(* IEC 61131-3 sources: nvidia-ai-factory-controls/libraries/AIFactory_Communication/POUs/Subscribers, 5 files *)

(* ---- FB_Subscriber_BACnet.fb ---- *)
(* =============================================================================
    FB_Subscriber_BACnet — BACnet/IP Client Subscriber
    Common Library | NVIDIA AI Factory Controls
   =============================================================================

   PURPOSE:
     Implements I_DataSubscriber by reading BACnet objects from external
     BMS/HVAC controllers. Used to collect:
       • Ambient temperature from building sensors
       • Outdoor wet-bulb temperature (for economizer decisions)
       • HVAC status (AHU running, damper positions)
       • Chilled water supply temperature from central plant
       • Building fire alarm status (BACnet notification class)

   POLLING MODEL:
     Similar to Modbus subscriber: maintains a poll table of
     BACnet ReadProperty requests. Cycles through in round-robin.

   BACnet SERVICES USED:
     • ReadProperty (single object read)
     • ReadPropertyMultiple (batch read — more efficient)
     • SubscribeCOV (Change-of-Value subscription — event-driven)

   COV (Change-of-Value):
     For critical values (fire alarm, ambient temp), use COV subscription
     instead of polling. BACnet server pushes changes immediately.
     Reduces latency from poll-interval to near-real-time.

   REQUIRES:
     CODESYS BACnet/IP Client device in project tree.
     Or: BACnet client library.

   THREAD SAFETY:
     Runs in Communication_Task. BACnet I/O is handled by CODESYS
     BACnet stack asynchronously; this FB reads the results.
   ============================================================================= *)

(* ═══════════════════════════════════════════════════════════════════════════════
   DECLARATION
   ═══════════════════════════════════════════════════════════════════════════════ *)

FUNCTION_BLOCK FB_Subscriber_BACnet IMPLEMENTS I_DataSubscriber
VAR_INPUT
    (* --- Timing --- *)
    fCycleTime_s         : REAL := 0.1;
    nMaxPollsPerCycle    : USINT := 4;
    nStaleTimeout_ms     : UDINT := 10000;

    (* --- COV Configuration --- *)
    bUseCOV              : BOOL := TRUE;    (* Prefer COV over polling *)
    nCOV_Lifetime_s      : UDINT := 300;    (* COV subscription lifetime *)
END_VAR

VAR
    _bConnected          : BOOL;
    _nSubscriptionCount  : UDINT;
    _nStaleCount         : UDINT;

    (* --- Poll Request Table --- *)
    _astPollRequests     : ARRAY[1..32] OF ST_BACnetPollRequest;
    _nPollCount          : USINT;
    _nCurrentPoll        : USINT;

    (* --- COV Subscriptions --- *)
    _astCOV_Subs         : ARRAY[1..16] OF ST_BACnetCOVSub;
    _nCOV_Count          : USINT;

    (* --- Received Data --- *)
    _astReceivedData     : ARRAY[1..64] OF ST_Subscription;
    _nReceivedCount      : UINT;

    (* --- Discovered Values (commonly needed) --- *)
    fAmbientTemp         : REAL;            (* Outdoor ambient temperature [°C] *)
    fWetBulbTemp         : REAL;            (* Wet-bulb temperature [°C] *)
    fCHW_SupplyTemp      : REAL;            (* Chilled water supply [°C] *)
    bBuildingFireAlarm   : BOOL;            (* Building fire alarm active *)
    bAHU_Running         : ARRAY[1..4] OF BOOL;  (* Air handling unit status *)

    (* --- Statistics --- *)
    _nTotalReads         : UDINT;
    _nSuccessfulReads    : UDINT;
    _nCOV_Notifications  : UDINT;           (* COV events received *)

    (* --- Edge Triggers --- *)
    _rtrigFireAlarm      : R_TRIG;          (* Building fire alarm activated *)
    _ftrigFireAlarm      : F_TRIG;          (* Building fire alarm cleared *)
END_VAR

(* ═══════════════════════════════════════════════════════════════════════════════
   IMPLEMENTATION
   ═══════════════════════════════════════════════════════════════════════════════ *)

(* --- Fire Alarm Edge Detection --- *)
_rtrigFireAlarm(CLK := bBuildingFireAlarm);
_ftrigFireAlarm(CLK := bBuildingFireAlarm);

(* --- Round-Robin Polling (same pattern as Modbus subscriber) --- *)
(* In production with CODESYS BACnet library:
   FOR i := 1 TO nMaxPollsPerCycle DO
       _nCurrentPoll := _nCurrentPoll + 1;
       IF _nCurrentPoll > _nPollCount THEN _nCurrentPoll := 1; END_IF

       // Execute BACnet ReadProperty
       // Object: _astPollRequests[_nCurrentPoll].nObjectType
       // Instance: _astPollRequests[_nCurrentPoll].nObjectInstance
       // Property: Present_Value (85)

       // On success: store value, update timestamp
       // On error: increment error count
   END_FOR *)

(* --- COV Subscription Renewal --- *)
(* BACnet COV subscriptions expire. Renew before lifetime expires.
   In production: check each _astCOV_Subs lifetime remaining,
   re-subscribe if < 60 seconds remaining. *)

(* --- Stale Detection --- *)
_nStaleCount := 0;
(* Check all subscriptions for staleness *)

(* ---- FB_Subscriber_Modbus.fb ---- *)
(* =============================================================================
    FB_Subscriber_Modbus — Modbus TCP Master (Client) Subscriber
    Common Library | NVIDIA AI Factory Controls
   =============================================================================

   PURPOSE:
     Implements I_DataSubscriber by polling Modbus TCP slave devices.
     Used to collect data from:
       • Energy meters (Schneider PM5xxx, ABB M4M)
       • UPS systems (Vertiv/Eaton Modbus interface)
       • PDU intelligent panels
       • CDU controllers (if not on EtherCAT)
       • ATS controllers

   POLLING MODEL:
     Maintains a list of Modbus read requests (device, register, count).
     Cycles through requests in round-robin fashion.
     Each poll result is stored with timestamp for freshness tracking.

   REGISTER INTERPRETATION:
     • Holding Registers (FC03): most common for read data
     • Input Registers (FC04): read-only process values
     • REAL values: 2 consecutive registers, IEEE 754 float (big-endian)
     • BOOL values: individual bits within a register (coils FC01)

   REQUIRES:
     CODESYS Modbus TCP Master device in project tree.
     Or: ModbusFB library (Modbus.ModbusTCPMaster)

   PERFORMANCE:
     At 100ms cycle, one poll per scan = 10 polls/s per device.
     With 5 devices × 10 registers each = can poll all within 5 seconds.
     Configurable: nMaxPollsPerCycle controls throughput.
   ============================================================================= *)

(* ═══════════════════════════════════════════════════════════════════════════════
   DECLARATION
   ═══════════════════════════════════════════════════════════════════════════════ *)

FUNCTION_BLOCK FB_Subscriber_Modbus IMPLEMENTS I_DataSubscriber
VAR_INPUT
    (* --- Timing --- *)
    fCycleTime_s         : REAL := 0.1;
    nMaxPollsPerCycle    : USINT := 2;      (* Max Modbus transactions per scan *)
    nStaleTimeout_ms     : UDINT := 5000;   (* 5s without response = stale *)
END_VAR

VAR
    _bConnected          : BOOL := TRUE;    (* "Connected" if any device responding *)
    _nSubscriptionCount  : UDINT;
    _nStaleCount         : UDINT;

    (* --- Poll Request Table --- *)
    _astPollRequests     : ARRAY[1..32] OF ST_ModbusPollRequest;
    _nPollCount          : USINT;
    _nCurrentPoll        : USINT;           (* Round-robin index *)

    (* --- Received Data --- *)
    _astReceivedData     : ARRAY[1..64] OF ST_Subscription;
    _nReceivedCount      : UINT;

    (* --- Device Connection Tracking --- *)
    _abDeviceAlive       : ARRAY[1..8] OF BOOL;   (* Per-device health *)
    _anDeviceErrors      : ARRAY[1..8] OF UINT;   (* Consecutive errors *)
    _nMaxErrors          : UINT := 5;              (* Errors before marking dead *)

    (* --- Statistics --- *)
    _nTotalPolls         : UDINT;
    _nSuccessfulPolls    : UDINT;
    _nTimeoutErrors      : UDINT;

    (* --- Edge Triggers --- *)
    _rtrigDeviceLost     : ARRAY[1..8] OF F_TRIG;  (* Device went offline *)
END_VAR

(* ═══════════════════════════════════════════════════════════════════════════════
   IMPLEMENTATION
   ═══════════════════════════════════════════════════════════════════════════════ *)

(* --- Round-Robin Polling --- *)
(* Each scan, execute up to nMaxPollsPerCycle Modbus read operations.
   Advance _nCurrentPoll to next request. Skip devices marked dead. *)

(* In production with CODESYS Modbus library:
   FOR i := 1 TO nMaxPollsPerCycle DO
       _nCurrentPoll := _nCurrentPoll + 1;
       IF _nCurrentPoll > _nPollCount THEN _nCurrentPoll := 1; END_IF

       IF _abDeviceAlive[_astPollRequests[_nCurrentPoll].nDeviceID] THEN
           // Execute Modbus FC03 read
           // On success: update _astReceivedData, reset error count
           // On timeout: increment error count, mark dead if > _nMaxErrors
       END_IF
   END_FOR *)

(* --- Stale Detection --- *)
_nStaleCount := 0;
(* Check each subscription's age vs timeout *)

(* --- Connection Status --- *)
_bConnected := FALSE;
(* If ANY device is alive, we're "connected" *)

(* ---- FB_Subscriber_MQTT.fb ---- *)
(* =============================================================================
    FB_Subscriber_MQTT — MQTT Data Subscriber
    Common Library | NVIDIA AI Factory Controls
   =============================================================================

   PURPOSE:
     Implements I_DataSubscriber for receiving data via MQTT.
     Used for:
       • Cloud commands (setpoint changes from SCADA/DCIM)
       • GPU telemetry (DCGM data published by edge gateway)
       • Inter-site data exchange
       • Digital twin commands (Omniverse → PLC)

   TOPIC STRUCTURE:
     Subscribe topics configured as array. Supports wildcards:
       'aifactory/+/cmd/#'        — All commands for this site
       'gpu/+/telemetry'          — GPU telemetry from all racks
       'cloud/setpoints/cooling'  — Cloud-issued cooling setpoints

   PAYLOAD FORMAT:
     JSON: {"value": 35.2, "quality": 0, "timestamp": 1717000000000}
     Or Sparkplug B binary (decoded by MQTT library)

   REQUIRES:
     CODESYS IoT MQTT library (IoDrvMQTTClient or MQTT.MQTTClient)

   THREAD SAFETY:
     Runs in Communication_Task only. Received values stored in
     internal buffer, copied to GVL_CrossTask at end of cycle.
   ============================================================================= *)

(* ═══════════════════════════════════════════════════════════════════════════════
   DECLARATION
   ═══════════════════════════════════════════════════════════════════════════════ *)

FUNCTION_BLOCK FB_Subscriber_MQTT IMPLEMENTS I_DataSubscriber
VAR_INPUT
    (* --- Broker Configuration --- *)
    sBrokerURL           : STRING(128) := 'tcp://192.168.200.10:1883';
    sClientID            : STRING(64) := 'IPC-02-SUB';
    sUsername            : STRING(64) := '';
    sPassword            : STRING(64) := '';
    bUseTLS              : BOOL := FALSE;

    (* --- Subscription Topics (up to 16) --- *)
    asTopics             : ARRAY[1..16] OF STRING(128);
    nTopicCount          : USINT := 0;

    (* --- QoS --- *)
    nQoS                 : USINT := 1;      (* 1 = at-least-once for commands *)

    (* --- Timing --- *)
    fCycleTime_s         : REAL := 0.1;
    nStaleTimeout_ms     : UDINT := 10000;  (* 10s without update = stale *)
END_VAR

VAR
    _bConnected          : BOOL;
    _nSubscriptionCount  : UDINT;
    _nStaleCount         : UDINT;

    (* --- Received Data Buffer --- *)
    (* Stores last received value per subscription path.
       Communication_Task reads these and writes to GVL_CrossTask. *)
    _astReceivedData     : ARRAY[1..64] OF ST_Subscription;
    _nReceivedCount      : UINT;

    (* --- Connection Management --- *)
    _tonReconnect        : TON;
    _tReconnectInterval  : TIME := T#5S;
    _bConnectRequested   : BOOL;
    _nReconnectAttempts  : UINT;

    (* --- Edge Triggers --- *)
    _rtrigConnected      : R_TRIG;          (* Connection established *)
    _ftrigDisconnected   : F_TRIG;          (* Connection lost *)

    (* --- Statistics --- *)
    _nMessagesReceived   : UDINT;           (* Total messages received *)
    _nParseErrors        : UDINT;           (* Messages that failed to parse *)
    _nLastReceiveTime_ms : UDINT;           (* Time of last message *)

    (* --- MQTT Client (from CODESYS IoT library) --- *)
    (* _fbMqttClient     : MQTT.MQTTClient;  -- uncomment when library imported *)
    (* _fbMqttSubscribe  : MQTT.MQTTSubscribe; *)
END_VAR

(* ═══════════════════════════════════════════════════════════════════════════════
   IMPLEMENTATION
   ═══════════════════════════════════════════════════════════════════════════════ *)

(* --- Edge detection on connection state --- *)
_rtrigConnected(CLK := _bConnected);
_ftrigDisconnected(CLK := _bConnected);

(* --- Reconnection logic --- *)
IF _bConnectRequested AND NOT _bConnected THEN
    _tonReconnect(IN := TRUE, PT := _tReconnectInterval);
    IF _tonReconnect.Q THEN
        _tonReconnect(IN := FALSE);
        _nReconnectAttempts := _nReconnectAttempts + 1;
        (* _fbMqttClient.Connect(sBrokerURL, sClientID, ...); *)
    END_IF
ELSE
    _tonReconnect(IN := FALSE);
END_IF

(* --- Stale detection: check all subscriptions --- *)
_nStaleCount := 0;
(* In production: iterate _astReceivedData, check age vs nStaleTimeout_ms *)

(* ---- FB_Subscriber_OPCUA.fb ---- *)
(* =============================================================================
    FB_Subscriber_OPCUA — OPC UA Client Subscriber
    Common Library | NVIDIA AI Factory Controls
   =============================================================================

   PURPOSE:
     Implements I_DataSubscriber using CODESYS OPC UA client.
     Reads data FROM external OPC UA servers:
       • Other IPCs (IPC-01 reading safety status from IPC-04)
       • Edge gateway (GPU telemetry exposed via OPC UA)
       • Third-party equipment (CDU controllers, UPS, PDU)

   USE CASE:
     • Inter-IPC data exchange (OPC UA is the primary protocol)
     • Reading GPU telemetry from edge gateway
     • Collecting data from BMS/DCIM systems

   CONNECTION MODEL:
     CODESYS OPC UA Client device is added in the project tree.
     Variables are mapped in the Symbol Configuration of the client device.
     This FB wraps that mechanism with the I_DataSubscriber interface.

   FRESHNESS MONITORING:
     Each subscribed variable tracks its last-update time.
     If a variable hasn't updated within expected interval × 3, it's
     marked as STALE. Consumer logic can then use fallback values.

   REQUIRES:
     CODESYS OPC UA Client device in project (CmpOPCUAClient).
   ============================================================================= *)

(* ═══════════════════════════════════════════════════════════════════════════════
   DECLARATION
   ═══════════════════════════════════════════════════════════════════════════════ *)

FUNCTION_BLOCK FB_Subscriber_OPCUA IMPLEMENTS I_DataSubscriber
VAR_INPUT
    (* --- Connection Configuration --- *)
    sServerURL           : STRING(128) := 'opc.tcp://192.168.100.100:4840';
    sServerName          : STRING(64) := 'EdgeGateway';
    nReconnectInterval_s : UINT := 5;
    nDefaultTimeout_ms   : UDINT := 5000;
END_VAR

VAR
    _bConnected          : BOOL;
    _nSubscriptionCount  : UDINT;
    _nStaleCount         : UDINT;

    (* Subscription tracking *)
    _astSubscriptions    : ARRAY[1..100] OF ST_Subscription;
    _nSubCount           : UINT;

    (* Connection management *)
    _tonReconnect        : TON;
    _bReconnecting       : BOOL;
END_VAR

(* ═══════════════════════════════════════════════════════════════════════════════
   IMPLEMENTATION
   ═══════════════════════════════════════════════════════════════════════════════ *)

(* OPC UA client connection management.
   In CODESYS, the OPC UA Client device handles connection automatically.
   This FB monitors the connection state and tracks data freshness. *)

(* Check for stale subscriptions *)
_nStaleCount := 0;
(* Would iterate _astSubscriptions and check age vs. expected interval *)

(* ---- FB_Subscriber_REST.fb ---- *)
(* =============================================================================
    FB_Subscriber_REST — HTTP/REST Client for GPU Telemetry (DCGM)
    Common Library | NVIDIA AI Factory Controls
   =============================================================================

   PURPOSE:
     Implements I_DataSubscriber by polling REST API endpoints.
     Primary use case: reading NVIDIA DCGM (Data Center GPU Manager) data.

   GPU TELEMETRY ENDPOINT:
     DCGM exposes metrics at: http://{host}:9400/metrics (Prometheus format)
     Or via gRPC/REST: http://{host}:5555/v1/gpu/status

   DATA COLLECTED:
     • GPU junction temperature (per GPU)
     • GPU power draw (per GPU)
     • GPU utilization (%)
     • Memory temperature
     • NVLink bandwidth utilization
     • Thermal throttle status

   ARCHITECTURE:
     This FB does NOT make HTTP calls directly from CODESYS.
     Instead, the edge gateway Python service polls DCGM and publishes
     results to OPC UA or MQTT. This FB reads from that intermediate layer.

     Alternative (direct from CODESYS):
       Uses CODESYS SysSocket + HTTP client library for direct REST calls.
       Only feasible on x86 IPCs with sufficient resources.

   POLLING STRATEGY:
     • Poll interval: 1-10 seconds (configurable)
     • Timeout: 2 seconds per request
     • On timeout: mark data stale, use last-known-good values
     • On 3 consecutive timeouts: mark device offline

   REQUIRES:
     CODESYS HTTP Client library (CmpWebClient or SysSocket raw)
     OR: edge gateway intermediate translation (preferred)

   THREAD SAFETY:
     HTTP operations are blocking. Run at low priority (Communication_Task).
     Never block the Control_Task or Safety_Task.
   ============================================================================= *)

(* ═══════════════════════════════════════════════════════════════════════════════
   DECLARATION
   ═══════════════════════════════════════════════════════════════════════════════ *)

FUNCTION_BLOCK FB_Subscriber_REST IMPLEMENTS I_DataSubscriber
VAR_INPUT
    (* --- Endpoint Configuration --- *)
    sBaseURL             : STRING(128) := 'http://192.168.200.50:9400';
    sEndpointPath        : STRING(64) := '/metrics';
    nPollInterval_ms     : UDINT := 2000;   (* Poll every 2 seconds *)
    nTimeout_ms          : UDINT := 2000;   (* HTTP timeout *)

    (* --- Authentication (if required) --- *)
    sAuthToken           : STRING(128) := '';
    bUseAuth             : BOOL := FALSE;

    (* --- Timing --- *)
    fCycleTime_s         : REAL := 0.1;
END_VAR

VAR
    _bConnected          : BOOL;
    _nSubscriptionCount  : UDINT;
    _nStaleCount         : UDINT;

    (* --- Poll Timing --- *)
    _nTimeSinceLastPoll  : UDINT;
    _bPollPending        : BOOL;

    (* --- Response Parsing --- *)
    _sLastResponse       : STRING(4096);    (* Last HTTP response body *)
    _bResponseValid      : BOOL;

    (* --- GPU Data (parsed from response) --- *)
    _afGPU_Temperature   : ARRAY[1..72] OF REAL;   (* Per-GPU temp [°C] *)
    _afGPU_Power         : ARRAY[1..72] OF REAL;   (* Per-GPU power [W] *)
    _afGPU_Utilization   : ARRAY[1..72] OF REAL;   (* Per-GPU util [%] *)
    _nGPU_Count          : USINT;                  (* Detected GPU count *)
    _fGPU_MaxTemp        : REAL;                   (* Max across all GPUs *)
    _fGPU_TotalPower_kW  : REAL;                   (* Sum of all GPU power *)

    (* --- Health Tracking --- *)
    _nConsecutiveErrors  : USINT;
    _nMaxErrors          : USINT := 3;
    _nTotalRequests      : UDINT;
    _nSuccessfulRequests : UDINT;

    (* --- Edge Triggers --- *)
    _rtrigPollDue        : R_TRIG;          (* Time to poll *)
    _ftrigConnectionLost : F_TRIG;          (* Connection went down *)

    (* --- Received Data (I_DataSubscriber interface) --- *)
    _astReceivedData     : ARRAY[1..32] OF ST_Subscription;
    _nReceivedCount      : UINT;
END_VAR

(* ═══════════════════════════════════════════════════════════════════════════════
   IMPLEMENTATION
   ═══════════════════════════════════════════════════════════════════════════════ *)

(* --- Poll Timing --- *)
_nTimeSinceLastPoll := _nTimeSinceLastPoll + REAL_TO_UDINT(fCycleTime_s * 1000.0);
_bPollPending := (_nTimeSinceLastPoll >= nPollInterval_ms);

IF _bPollPending AND NOT _bPollPending THEN
    (* In production with CODESYS HTTP library:
       1. Build HTTP GET request to sBaseURL + sEndpointPath
       2. Add auth header if bUseAuth
       3. Send request (async or sync depending on library)
       4. On response: parse JSON/Prometheus format
       5. Extract GPU temps, power, utilization
       6. Update _afGPU_* arrays
       7. Calculate _fGPU_MaxTemp, _fGPU_TotalPower_kW
       8. Update _astReceivedData for I_DataSubscriber consumers
       9. Reset _nTimeSinceLastPoll
       10. On error: increment _nConsecutiveErrors *)
    _nTimeSinceLastPoll := 0;
    _nTotalRequests := _nTotalRequests + 1;
END_IF

(* --- Connection Status --- *)
_ftrigConnectionLost(CLK := _bConnected);
_bConnected := (_nConsecutiveErrors < _nMaxErrors);

(* --- Aggregate GPU Metrics --- *)
(* In production: scan _afGPU_Temperature for max, sum _afGPU_Power *)
